// TwinCAT 3 PLC project PlcLibrary1
// Title: PlcLibrary1
// Company: My Company
// ProjectVersion: 1.2.3.4
// ProgramVersion: 3.1.4024.0
// libraries:
//   Tc2_Standard, * (Beckhoff Automation GmbH)
//   Tc2_System, * (Beckhoff Automation GmbH)
// project tree:
//   POUs/ MAIN.TcPOU

// ---- POUs/MAIN.TcPOU
PROGRAM MAIN
VAR
END_VAR

END_PROGRAM
